PROGRAM QRob_StateMachine
VAR_INPUT
init_: BOOL:= True;
//global aux state
G_STATE : INT := -1;
//comaper position to stop
Position : LREAL:= 0;
Velocity : REAL:=170;
Torque : INT := 0;
Torque_ramp : INT := 100;
Control :E_DRIVEOPERATIONMODE;
Reset_State : BOOL:= FALSE;
//Max_profile_velocity AT%Q*:UDINT := 314572;
//Modes_operation AT%Q*:USINT:= 8;
//actual_torque AT%I*:INT ;

//Qrob_set torque 
torquevalut AT%Q*:INT;


END_VAR
VAR_OUTPUT
	State_complete : BOOL := FALSE;
	Act_Gl_State : INT := -1;
	Act_In_State : INT := -1;
	Act_Pos : LREAL := -1;
END_VAR
VAR
	
//Axis status
Axis_state :BOOL:=FALSE;
	//internal aux state
I_STATE : INT:=-1;
Aux_error :INT:=-1;
//blocks to activate axis of qrob
Reset : MC_Reset;
ResetOut: ST_McOutputs;

PowerAxis1 : MC_Power;
/// debug function block output data 
PowerAxis1Out: ST_McOutputs;



//blocks to move axis 
MoveAbsAxis1 :MC_MoveAbsolute;
MoveAbsoluteOut1: ST_McOutputs;

//block to set home position
Home : MC_Home;
HomeOut: ST_McOutputs;

//block to read and change the contyrol mode
WriteDriveOperationMode : MC_WriteDriveOperationMode;
WDO_ModeOut : ST_McOutputs;

ReadDriveOperationMode : MC_ReadDriveOperationMode;
RDO_ModeOut : ST_McOutputs;
ReadOperation_mode : E_DRIVEOPERATIONMODE;

//block to Control Mode
TorqueControl : MC_TorqueControl;
TorqueControlOut : ST_McOutputs;
Torque_done : BOOL;
Qrob_velocity AT%I*:DINT := -1;
Qrob_torque AT%I*:INT := -1;

//block stop motion
Stop : MC_Stop;
StopOut: ST_McOutputs;

//var to ck torque done
F_vel : BOOL ;
F_tor : BOOL;
F_tor_done : BOOL;


//var to offfset Home
offset_home :INT := 3;
offset_flag : INT := -1;

Sensor_Position_detection AT%I*: BOOL;


END_VAR

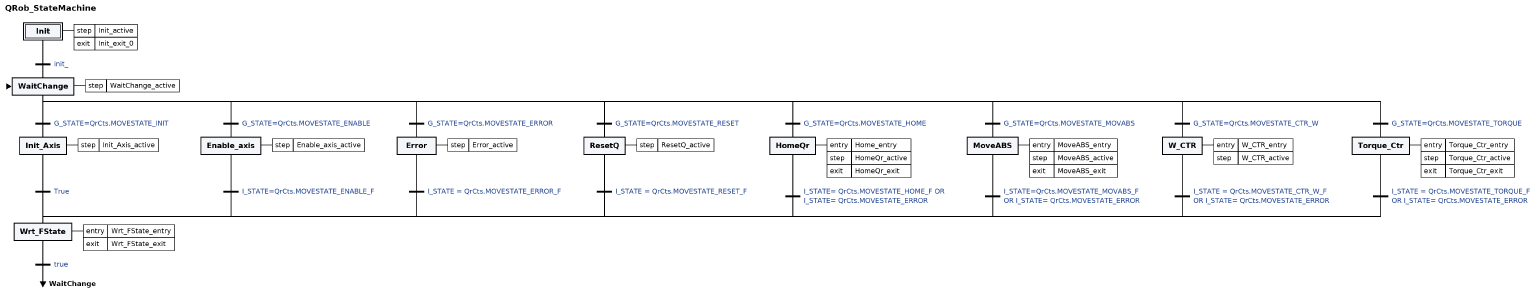
INITIAL_STEP Init:
    Init_active(N);  // step action
    Init_exit_0(P0);  // exit action
END_STEP
TRANSITION FROM Init TO WaitChange
    := init_;
END_TRANSITION
STEP WaitChange:
    WaitChange_active(N);  // step action
END_STEP
TRANSITION FROM WaitChange TO Init_Axis
    := G_STATE=QrCts.MOVESTATE_INIT;
END_TRANSITION
STEP Init_Axis:
    Init_Axis_active(N);  // step action
END_STEP
TRANSITION FROM Init_Axis TO Wrt_FState
    := True;
END_TRANSITION
TRANSITION FROM WaitChange TO Enable_axis
    := G_STATE=QrCts.MOVESTATE_ENABLE;
END_TRANSITION
STEP Enable_axis:
    Enable_axis_active(N);  // step action
END_STEP
TRANSITION FROM Enable_axis TO Wrt_FState
    := I_STATE=QrCts.MOVESTATE_ENABLE_F;
END_TRANSITION
TRANSITION FROM WaitChange TO Error
    := G_STATE=QrCts.MOVESTATE_ERROR;
END_TRANSITION
STEP Error:
    Error_active(N);  // step action
END_STEP
TRANSITION FROM Error TO Wrt_FState
    := I_STATE = QrCts.MOVESTATE_ERROR_F;
END_TRANSITION
TRANSITION FROM WaitChange TO ResetQ
    := G_STATE=QrCts.MOVESTATE_RESET;
END_TRANSITION
STEP ResetQ:
    ResetQ_active(N);  // step action
END_STEP
TRANSITION FROM ResetQ TO Wrt_FState
    := I_STATE = QrCts.MOVESTATE_RESET_F;
END_TRANSITION
TRANSITION FROM WaitChange TO HomeQr
    := G_STATE=QrCts.MOVESTATE_HOME;
END_TRANSITION
STEP HomeQr:
    Home_entry(P1);  // entry action
    HomeQr_active(N);  // step action
    HomeQr_exit(P0);  // exit action
END_STEP
TRANSITION FROM HomeQr TO Wrt_FState
    := I_STATE= QrCts.MOVESTATE_HOME_F OR I_STATE= QrCts.MOVESTATE_ERROR;
END_TRANSITION
TRANSITION FROM WaitChange TO MoveABS
    := G_STATE=QrCts.MOVESTATE_MOVABS;
END_TRANSITION
STEP MoveABS:
    MoveABS_entry(P1);  // entry action
    MoveABS_active(N);  // step action
    MoveABS_exit(P0);  // exit action
END_STEP
TRANSITION FROM MoveABS TO Wrt_FState
    := I_STATE=QrCts.MOVESTATE_MOVABS_F OR I_STATE= QrCts.MOVESTATE_ERROR;
END_TRANSITION
TRANSITION FROM WaitChange TO W_CTR
    := G_STATE=QrCts.MOVESTATE_CTR_W;
END_TRANSITION
STEP W_CTR:
    W_CTR_entry(P1);  // entry action
    W_CTR_active(N);  // step action
END_STEP
TRANSITION FROM W_CTR TO Wrt_FState
    := I_STATE = QrCts.MOVESTATE_CTR_W_F OR I_STATE= QrCts.MOVESTATE_ERROR;
END_TRANSITION
TRANSITION FROM WaitChange TO Torque_Ctr
    := G_STATE=QrCts.MOVESTATE_TORQUE;
END_TRANSITION
STEP Torque_Ctr:
    Torque_Ctr_entry(P1);  // entry action
    Torque_Ctr_active(N);  // step action
    Torque_Ctr_exit(P0);  // exit action
END_STEP
TRANSITION FROM Torque_Ctr TO Wrt_FState
    := I_STATE = QrCts.MOVESTATE_TORQUE_F OR I_STATE= QrCts.MOVESTATE_ERROR;
END_TRANSITION
STEP Wrt_FState:
    Wrt_FState_entry(P1);  // entry action
    Wrt_FState_exit(P0);  // exit action
END_STEP
TRANSITION FROM Wrt_FState TO WaitChange
    := true;
END_TRANSITION

ACTION AC_WriteControl:
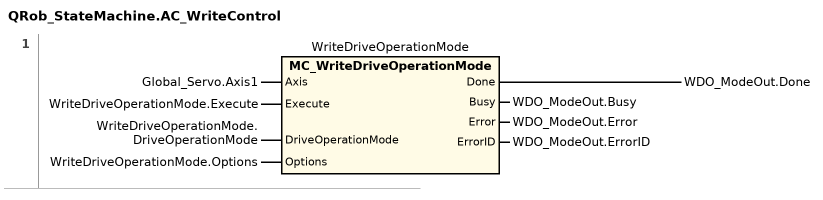
// NETWORK 1
WriteDriveOperationMode(
    Axis := Global_Servo.Axis1,
    Execute := WriteDriveOperationMode.Execute,
    DriveOperationMode := WriteDriveOperationMode.DriveOperationMode,
    Options := WriteDriveOperationMode.Options,
    Busy => WDO_ModeOut.Busy,
    Error => WDO_ModeOut.Error,
    ErrorID => WDO_ModeOut.ErrorID); // MC_WriteDriveOperationMode
WDO_ModeOut.Done := WriteDriveOperationMode.Done;
END_ACTION

ACTION Act_Home:
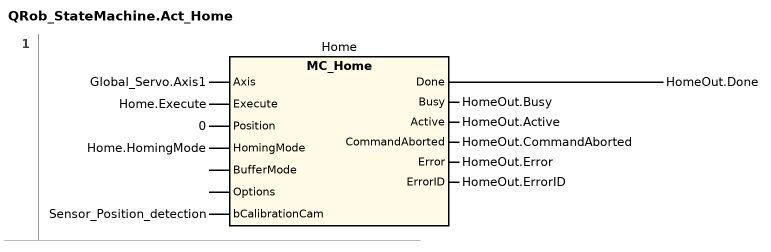
// NETWORK 1
Home(
    Axis := Global_Servo.Axis1,
    Execute := Home.Execute,
    Position := 0,
    HomingMode := Home.HomingMode,
    bCalibrationCam := Sensor_Position_detection,
    Busy => HomeOut.Busy,
    Active => HomeOut.Active,
    CommandAborted => HomeOut.CommandAborted,
    Error => HomeOut.Error,
    ErrorID => HomeOut.ErrorID); // MC_Home
HomeOut.Done := Home.Done;
END_ACTION

ACTION Act_MoveAbs:
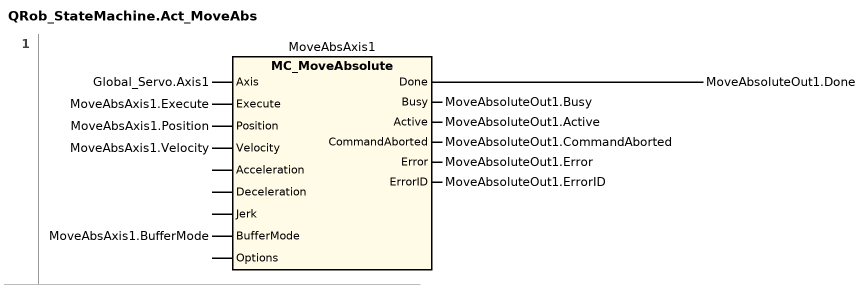
// NETWORK 1
MoveAbsAxis1(
    Axis := Global_Servo.Axis1,
    Execute := MoveAbsAxis1.Execute,
    Position := MoveAbsAxis1.Position,
    Velocity := MoveAbsAxis1.Velocity,
    BufferMode := MoveAbsAxis1.BufferMode,
    Busy => MoveAbsoluteOut1.Busy,
    Active => MoveAbsoluteOut1.Active,
    CommandAborted => MoveAbsoluteOut1.CommandAborted,
    Error => MoveAbsoluteOut1.Error,
    ErrorID => MoveAbsoluteOut1.ErrorID); // MC_MoveAbsolute
MoveAbsoluteOut1.Done := MoveAbsAxis1.Done;
END_ACTION

ACTION Act_Power:
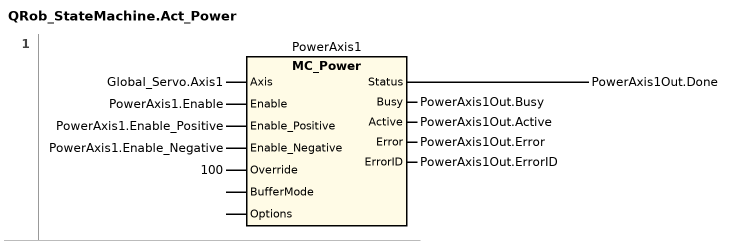
// NETWORK 1
PowerAxis1(
    Axis := Global_Servo.Axis1,
    Enable := PowerAxis1.Enable,
    Enable_Positive := PowerAxis1.Enable_Positive,
    Enable_Negative := PowerAxis1.Enable_Negative,
    Override := 100,
    Busy => PowerAxis1Out.Busy,
    Active => PowerAxis1Out.Active,
    Error => PowerAxis1Out.Error,
    ErrorID => PowerAxis1Out.ErrorID); // MC_Power
PowerAxis1Out.Done := PowerAxis1.Status;
END_ACTION

ACTION Act_ReadControl:
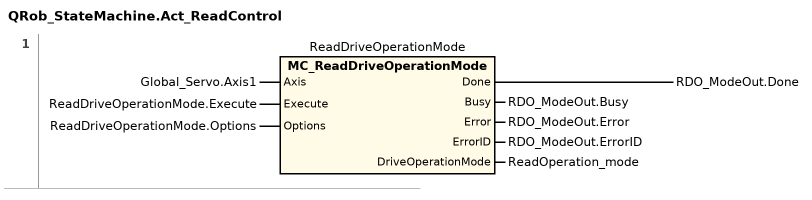
// NETWORK 1
ReadDriveOperationMode(
    Axis := Global_Servo.Axis1,
    Execute := ReadDriveOperationMode.Execute,
    Options := ReadDriveOperationMode.Options,
    Busy => RDO_ModeOut.Busy,
    Error => RDO_ModeOut.Error,
    ErrorID => RDO_ModeOut.ErrorID,
    DriveOperationMode => ReadOperation_mode); // MC_ReadDriveOperationMode
RDO_ModeOut.Done := ReadDriveOperationMode.Done;
END_ACTION

ACTION Act_Reset:
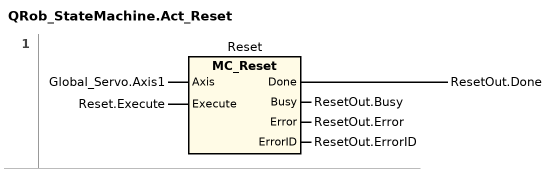
// NETWORK 1
Reset(
    Axis := Global_Servo.Axis1,
    Execute := Reset.Execute,
    Busy => ResetOut.Busy,
    Error => ResetOut.Error,
    ErrorID => ResetOut.ErrorID); // MC_Reset
ResetOut.Done := Reset.Done;
END_ACTION

ACTION Act_Stop:
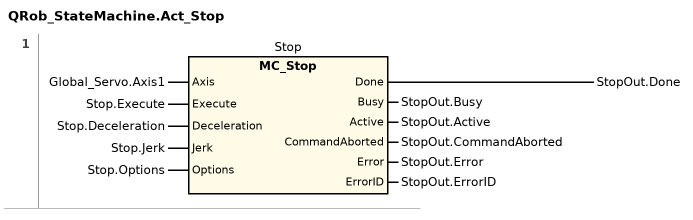
// NETWORK 1
Stop(
    Axis := Global_Servo.Axis1,
    Execute := Stop.Execute,
    Deceleration := Stop.Deceleration,
    Jerk := Stop.Jerk,
    Options := Stop.Options,
    Busy => StopOut.Busy,
    Active => StopOut.Active,
    CommandAborted => StopOut.CommandAborted,
    Error => StopOut.Error,
    ErrorID => StopOut.ErrorID); // MC_Stop
StopOut.Done := Stop.Done;
END_ACTION

ACTION Act_Torque:
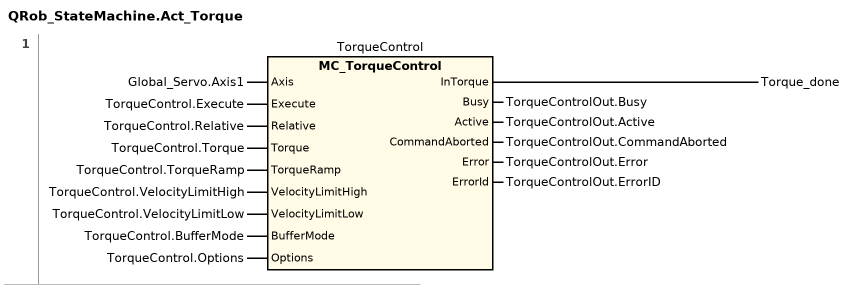
// NETWORK 1
TorqueControl(
    Axis := Global_Servo.Axis1,
    Execute := TorqueControl.Execute,
    Relative := TorqueControl.Relative,
    Torque := TorqueControl.Torque,
    TorqueRamp := TorqueControl.TorqueRamp,
    VelocityLimitHigh := TorqueControl.VelocityLimitHigh,
    VelocityLimitLow := TorqueControl.VelocityLimitLow,
    BufferMode := TorqueControl.BufferMode,
    Options := TorqueControl.Options,
    Busy => TorqueControlOut.Busy,
    Active => TorqueControlOut.Active,
    CommandAborted => TorqueControlOut.CommandAborted,
    Error => TorqueControlOut.Error,
    ErrorId => TorqueControlOut.ErrorID); // MC_TorqueControl
Torque_done := TorqueControl.InTorque;
END_ACTION

ACTION Enable_axis_active:
//power on axis
PowerAxis1.Enable := TRUE;
PowerAxis1.Enable_Positive := TRUE;
PowerAxis1.Enable_Negative := TRUE;


IF PowerAxis1.Status THEN
//check the state where the error is produced	
	CASE Aux_error OF 
		QrCts.MOVESTATE_MOVABS:
			G_STATE := QrCts.MOVESTATE_MOVABS;
		QrCts.MOVESTATE_HOME:
			G_STATE := QrCts.MOVESTATE_HOME;
		QrCts.MOVESTATE_CTR_W:
			G_STATE := QrCts.MOVESTATE_CTR_W;
		QrCts.MOVESTATE_TORQUE:	
			G_STATE := QrCts.MOVESTATE_TORQUE;
		QrCts.MOVESTATE_RELIEF:
			G_STATE := QrCts.MOVESTATE_RELIEF;
	ELSE
		G_STATE := -1;
	END_CASE
	I_STATE := QrCts.MOVESTATE_ENABLE_F;
ELSIF PowerAxis1.Error THEN
	G_STATE := QrCts.MOVESTATE_ERROR;
	I_STATE := QrCts.MOVESTATE_ENABLE_F;
END_IF

(* call the power function block *)
Act_Power();
Act_Reset();
Act_MoveAbs();
END_ACTION

ACTION Enable_axis_entry:
//power on axis
PowerAxis1.Enable := TRUE;
PowerAxis1.Enable_Positive := TRUE;
PowerAxis1.Enable_Negative := TRUE;
END_ACTION

ACTION Error_active:
IF Global_Servo.Axis1.NcToPlc.ErrorCode <>0 THEN
	G_STATE := QrCts.MOVESTATE_RESET;	(* axis error requires reset *)
	I_STATE := QrCts.MOVESTATE_ERROR_F;
ELSE
G_STATE := QrCts.MOVESTATE_INIT;
I_STATE := QrCts.MOVESTATE_ERROR_F;		(* function block errors don't need a reset *)
END_IF


(* call the power function block *)
Act_Power();
Act_Reset();
Act_MoveAbs();
END_ACTION

ACTION Home_entry:

//start fuction block 
Home.Execute := TRUE;

IF offset_flag = 1 THEN 
	Home.HomingMode := MC_Direct;
	offset_flag := offset_flag +1 ;
ELSE  	
	Home.HomingMode := MC_DefaultHoming;
END_IF


//write the retain state variable 
Act_Gl_State:=QrCts.MOVESTATE_HOME;
//read internal variable and write over output variable
I_STATE := QrCts.MOVESTATE_HOME_I;
Act_In_State := I_STATE;
END_ACTION

ACTION HomeQr_active:



//Home.bCalibrationCam := Sensor_Position_detection; 

IF Home.CommandAborted OR Home.Error THEN
	G_STATE := QrCts.MOVESTATE_ERROR;
	I_STATE := QrCts.MOVESTATE_ERROR;
	Aux_error := QrCts.MOVESTATE_HOME;
	Act_In_State := I_STATE;
ELSIF Home.Done THEN
	I_STATE := QrCts.MOVESTATE_HOME_F;
	//read internal variable and write over output variable
	Act_In_State := I_STATE;
	G_STATE := QrCts.MOVESTATE_MOVABS;
	position := offset_home;
	Home.Execute := FALSE; 
  IF offset_flag >= 2 THEN
	  G_STATE := -1;
	  offset_flag := -1;
  ELSE
	  G_STATE := QrCts.MOVESTATE_MOVABS;
	  offset_flag := offset_flag + 1;
  END_IF
	
END_IF





(* call the power function block *)
Act_Power();
Act_Reset();
Act_Home();
Act_MoveAbs();
END_ACTION

ACTION HomeQr_exit:
I_STATE :=-1;
END_ACTION

ACTION Init_active:

END_ACTION

ACTION Init_Axis_active:


//star variables
MoveAbsAxis1.Execute := FALSE;
Reset.Execute := FALSE;
Home.Execute := FALSE;
//write the global staus
G_State := QrCts.MOVESTATE_ENABLE;




(* call the power function block *)
Act_Power();
Act_Reset();
Act_MoveAbs();
Act_Home();
END_ACTION

ACTION Init_Axis_entry:

END_ACTION

ACTION Init_Axis_exit:

END_ACTION

ACTION Init_exit:
// NETWORK 1
END_ACTION

ACTION Init_exit_0:
G_STATE:=QrCts.MOVESTATE_INIT;


//check is there are some error
IF Global_Servo.Axis1.NcToPlc.ErrorCode <>0 THEN
	G_STATE := QrCts.MOVESTATE_RESET;	(* axis error requires reset *)
	
//ELSE
//	G_STATE := QrCts.MOVESTATE_INIT;
//	I_STATE := QrCts.MOVESTATE_ERROR_F;		(* function block errors don't need a reset *)
END_IF
END_ACTION

ACTION MoveABS_active:


IF MoveAbsAxis1.CommandAborted OR MoveAbsAxis1.Error THEN
	G_STATE := QrCts.MOVESTATE_ERROR;
	I_STATE := QrCts.MOVESTATE_ERROR;
	Aux_error := QrCts.MOVESTATE_MOVABS;
	Position := Position - Act_Pos;
	//read internal variable and write over output variable
	Act_In_State := I_STATE;
ELSIF MoveAbsAxis1.Done THEN
	I_STATE := QrCts.MOVESTATE_MOVABS_F;
	//read internal variable and write over output variable
	Act_In_State := I_STATE;
	G_STATE := -1;
	MoveAbsAxis1.Execute := FALSE;
ELSIF Reset_state THEN
	I_STATE := QrCts.MOVESTATE_MOVABS_F;;
	Act_In_State := I_STATE;
	G_STATE := -1;
	
	Stop.Execute := TRUE;
    MoveAbsAxis1.Execute := FALSE;	
	Reset_state := FALSE;
END_IF


//read actual postion
Act_Pos := Global_Servo.Axis1.NcToPlc.ActPos;

(* call the power function block *)
Act_Power();
Act_Reset();
Act_MoveAbs();
Act_Stop();
END_ACTION

ACTION MoveABS_entry:

MoveAbsAxis1.Position := Position;
MoveAbsAxis1.Velocity := Velocity;
//MoveAbsAxis1.BufferMode := MC_Buffered;
MoveAbsAxis1.Execute := TRUE;



//write the retain state variable 
Act_Gl_State:=QrCts.MOVESTATE_MOVABS;
//read internal variable and write over output variable
I_STATE := QrCts.MOVESTATE_MOVABS_I;
Act_In_State := I_STATE;

(* call the power function block *)
Act_Power();
Act_Reset();
Act_MoveAbs();
Act_Stop();
END_ACTION

ACTION MoveABS_exit:

//condition to execute home position
IF offset_flag = 0 THEN 
	G_STATE := QrCts.MOVESTATE_HOME;
    offset_flag := offset_flag +1 ;
END_IF


I_STATE :=-1;


Stop.Execute := FALSE;
Reset_state := FALSE;


(* call the power function block *)
Act_Power();
Act_Reset();
Act_MoveAbs();
Act_Stop();
END_ACTION

ACTION ResetQ_active:
WriteDriveOperationMode.Execute := FALSE;
Home.Execute := FALSE;
ReadDriveOperationMode.Execute := FALSE;
Stop.Execute := FALSE;
MoveAbsAxis1.Execute := FALSE;
TorqueControl.Execute := FALSE;
Stop.Execute := FALSE; 

Reset.Execute := TRUE;


IF Reset.Done THEN
	G_STATE := QrCts.MOVESTATE_INIT;
	I_STATE := QrCts.MOVESTATE_RESET_F;
ELSIF Reset.Error THEN
	G_STATE := QrCts.MOVESTATE_INIT; (* can't do anything here *)
	//I_STATE := QrCts.MOVESTATE_RESET_F;
END_IF


(* call the power function block *)
Act_Power();
Act_Reset();
Act_MoveAbs();
Act_Stop();
END_ACTION

ACTION Sleep_exit:
TorqueControl.Execute := False;
END_ACTION

ACTION Torque_Ctr_active:
IF TorqueControlOut.CommandAborted OR TorqueControlOut.Error THEN
	G_STATE := QrCts.MOVESTATE_ERROR;
	I_STATE := QrCts.MOVESTATE_ERROR;
	Aux_error := QrCts.MOVESTATE_TORQUE;
	//read internal variable and write over output variable
	Act_In_State := I_STATE;
ELSIF Torque_done THEN
	F_tor_done := TRUE;
END_IF



IF Qrob_torque = Torque THEN 
	F_tor := TRUE;
		IF ABS(Qrob_velocity) <=60  THEN 
			F_vel := TRUE;
	END_IF
END_IF


IF F_vel AND F_tor AND F_tor_done THEN

	I_STATE := QrCts.MOVESTATE_TORQUE_F;
	//read internal variable and write over output variable
	Act_In_State := I_STATE;
	G_STATE := -1;
	TorqueControl.Execute := FALSE;
	Torque_done := FALSE;
	
	F_vel  := FALSE;
	F_tor  := FALSE;
	F_tor_done  := FALSE;
	//I_STATE :=-1;	

END_IF

(* call the power function block *)
Act_Power();
Act_Reset();
Act_MoveAbs();
Act_Torque();
END_ACTION

ACTION Torque_Ctr_entry:
// write the variables TorqueControl block function
TorqueControl.Relative := FALSE;
TorqueControl.Torque := Torque;
torquevalut := Torque;
TorqueControl.TorqueRamp := 100;
TorqueControl.VelocityLimitHigh := 100;
TorqueControl.VelocityLimitLow := 1;
TorqueControl.Execute := True;


//write the retain state variable 
Act_Gl_State:=QrCts.MOVESTATE_TORQUE;
//read internal variable and write over output variable
I_STATE := QrCts.MOVESTATE_TORQUE_I;
Act_In_State := I_STATE;
END_ACTION

ACTION Torque_Ctr_exit:
	TorqueControl.Execute := FALSE;
	Torque_done := FALSE;
	//I_STATE :=-1;
	//G_STATE := -1;
	
	I_STATE :=-1;
END_ACTION

ACTION Torque_Relie_active:
//ggggggggggggggg


IF TorqueControlOut.CommandAborted OR TorqueControlOut.Error THEN
	G_STATE := QrCts.MOVESTATE_ERROR;
	I_STATE := QrCts.MOVESTATE_ERROR;
	Aux_error := QrCts.MOVESTATE_RELIEF;
	//read internal variable and write over output variable
	Act_In_State := I_STATE;
ELSIF Torque_done THEN
	F_tor_done := TRUE;
END_IF

//F_tor_done := TRUE;

IF Qrob_torque = 0 THEN 
	F_tor := TRUE;
		IF (-5 <= Qrob_velocity) AND  (Qrob_velocity<= 5) THEN 
			F_vel := TRUE;
	END_IF
END_IF


IF F_vel AND F_tor AND F_tor_done THEN

	I_STATE := QrCts.MOVESTATE_RELIEF_F;
	//read internal variable and write over output variable
	Act_In_State := I_STATE;
	G_STATE := -1;
	TorqueControl.Execute := TRUE;
	Torque_done := FALSE;
	
	F_vel  := FALSE;
	F_tor  := FALSE;
	F_tor_done  := FALSE;
	//I_STATE :=-1;	

END_IF

(* call the power function block *)
Act_Power();
Act_Reset();
Act_MoveAbs();
Act_Torque();
END_ACTION

ACTION Torque_Relie_entry:
// write the variables TorqueControl block function
TorqueControl.Relative := FALSE;
TorqueControl.Torque := 0;
TorqueControl.TorqueRamp := 0;
TorqueControl.VelocityLimitHigh := 100;
TorqueControl.VelocityLimitLow := 0;
//torquevalut := 0;
TorqueControl.Execute := True;


//write the retain state variable 
Act_Gl_State:=QrCts.MOVESTATE_RELIEF;
//read internal variable and write over output variable
I_STATE := QrCts.MOVESTATE_RELIEF_I;
Act_In_State := I_STATE;
END_ACTION

ACTION Torque_Relie_exit:
	TorqueControl.Execute := FALSE;
	Torque_done := FALSE;
	
	I_STATE :=-1;
END_ACTION

ACTION W_CTR_active:
IF WriteDriveOperationMode.Error THEN
	G_STATE := QrCts.MOVESTATE_ERROR;
	I_STATE := QrCts.MOVESTATE_ERROR;
	Aux_error := QrCts.MOVESTATE_CTR_W;
	//read internal variable and write over output variable
	Act_In_State := I_STATE;
ELSIF WriteDriveOperationMode.Done THEN
	//Read if the control mode have been change
	ReadDriveOperationMode.Execute := TRUE;
	IF ReadDriveOperationMode.Error THEN
		G_STATE := QrCts.MOVESTATE_ERROR;
		I_STATE := QrCts.MOVESTATE_ERROR;
		Aux_error := QrCts.MOVESTATE_CTR_W;
		//read internal variable and write over output variable
		Act_In_State := I_STATE;
	 	ReadDriveOperationMode.Execute := FALSE; 
	
	ELSIF ReadDriveOperationMode.Done THEN
		
		IF ReadOperation_mode = Control THEN

			I_STATE := QrCts.MOVESTATE_CTR_W_F;
			//read internal variable and write over output variable
			Act_In_State := I_STATE;
			//G_STATE := -1;
			WriteDriveOperationMode.Execute := FALSE;
			ReadDriveOperationMode.Execute := FALSE; 
			G_STATE := QrCts.MOVESTATE_RESET;
			//I_STATE :=-1;
		END_IF
		ReadDriveOperationMode.Execute := FALSE; 
	END_IF
END_IF


(* call the  function block *)
Act_Power();
Act_Reset();
AC_WriteControl();
Act_ReadControl();
END_ACTION

ACTION W_CTR_entry:
WriteDriveOperationMode.DriveOperationMode := Control;
WriteDriveOperationMode.Execute := TRUE;

//write the retain state variable 
Act_Gl_State:=QrCts.MOVESTATE_CTR_W;
//read internal variable and write over output variable
I_STATE := QrCts.MOVESTATE_CTR_W_I;
Act_In_State := I_STATE;
END_ACTION

ACTION WaitChange_active:

END_ACTION

ACTION Wrt_FState_entry:
//write output variable to indicate that the robot execute the state 
State_complete := TRUE;
END_ACTION

ACTION Wrt_FState_exit:
//write output variable to indicate that the robot execute the state 
State_complete := FALSE;
Reset_State := FALSE;
END_ACTION

END_PROGRAM

(* stored: Version 1.1.0.1, ProductVersion 3.1.4024.4
   POU QRob_StateMachine: Id {dea1dd88-39fa-4c4e-93c5-ae49219992d0}, SpecialFunc None
   Folder FBD: Id {740e0444-8ebf-4807-b223-6740ed61f611}
   Action AC_WriteControl: Id {c634974a-3fc3-4c20-bf17-ebeb1b3c1bdb}
   Action Act_Home: Id {76b70dda-cd7f-475a-b235-791ab72c2a92}
   Action Act_MoveAbs: Id {6915af91-f4b1-4d40-99ec-2e82ddc50489}
   Action Act_Power: Id {85cbb579-2a28-41af-a636-5432fe4f3d32}
   Action Act_ReadControl: Id {3f4eba52-287f-41ef-b8ce-ea25e281c168}
   Action Act_Reset: Id {72bd7d89-8767-4432-9292-a02562910a3e}
   Action Act_Stop: Id {26505a23-4e44-45d0-9c77-b8833fb0c0ad}
   Action Act_Torque: Id {16c3413b-972a-48fa-80e9-14e85defe8c8}
   Action Enable_axis_active: Id {726fecb4-69c6-4e7e-b391-d74d063e5215}
   Action Enable_axis_entry: Id {7c08845f-6242-4a60-abce-092305ddb52c}
   Action Error_active: Id {aa255cf8-ca48-4d1d-8627-2660654bd901}
   Action Home_entry: Id {32fb9a46-1642-4fad-a483-bae60448ec3f}
   Action HomeQr_active: Id {b5618258-2f10-4510-a97f-b7baa41bad28}
   Action HomeQr_exit: Id {3fafbdf9-9d7f-430f-9083-ecea0f8230a3}
   Action Init_active: Id {4171cb51-6252-4852-8e5b-da3c7c8c4cab}
   Action Init_Axis_active: Id {608179b8-0262-4a68-a08f-58e80770ad5d}
   Action Init_Axis_entry: Id {5fd46cfc-1bd1-434f-9105-dd6f5ba24956}
   Action Init_Axis_exit: Id {abd3e983-30fb-4cee-b74a-8a6f429417e0}
   Action Init_exit: Id {3e8dc8b2-5964-4b3d-b8a0-3598d1ff1d70}
   Action Init_exit_0: Id {ed758feb-5b02-4375-b9ea-b9b9faee0165}
   Action MoveABS_active: Id {bf482580-bca4-4945-86ee-79bf57cd951e}
   Action MoveABS_entry: Id {9d94e85e-c06d-4c66-9245-d026bb8c50a7}
   Action MoveABS_exit: Id {8591755a-eb2f-49ed-a34a-97f8e644fc9b}
   Action ResetQ_active: Id {c6601bd5-2819-48da-a47b-7c01580c8bc3}
   Action Sleep_exit: Id {e5e02b0f-9c09-482f-8256-e8489562b757}
   Action Torque_Ctr_active: Id {6581ea3e-dcc0-4dca-af33-c9d0f91e2ffe}
   Action Torque_Ctr_entry: Id {002bc9a7-4a12-417b-8653-8946a673df29}
   Action Torque_Ctr_exit: Id {79f1846d-b8cc-416f-9c5c-730eebcf7d98}
   Action Torque_Relie_active: Id {3753c684-e6cc-40d3-9ef7-1eb3c390fee5}
   Action Torque_Relie_entry: Id {41b73ce4-e55a-4c8d-97ff-d2c04dba97f7}
   Action Torque_Relie_exit: Id {986f84d1-523e-4636-979e-01ae3240dc48}
   Action W_CTR_active: Id {d51b996f-f75e-45dc-af1d-900f0bdcc7c2}
   Action W_CTR_entry: Id {3af00088-387f-4293-b320-f96cc7413082}
   Action WaitChange_active: Id {5dd4c232-e59a-4523-b7b5-0efd86db45ae}
   Action Wrt_FState_entry: Id {3fbfb66e-3783-4488-abed-6480d2af081b}
   Action Wrt_FState_exit: Id {e2a5e084-3023-4a1d-a625-641239d53d18} *)
